ABB RobotStudio station: Solution59_1.rsstn

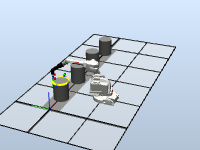
Station Solution59_1 (saved by RobotStudio format 3)
Controller IRB_52_1.20m, task T_ROB1: task frame (RAPID world) sits at (500, 0, 0) mm in the station
Controller IRB_52_1.20m
  mechanical unit CNV1: ?, 1 joints, base frame (0, 0, 0) mm
  mechanical unit ROB_1: IRB52_12_475_1005__01, 6 joints, base frame (500, -1000, 0) mm, rotated rx 0 ry 0 rz 90 deg
Layout (positions relative to the parent item):
  - IRB52_12_475_1005__01 [mechanism, from Robots\IRB52_12_475_1005_G_01.rslib] at (1000, -1000, 0) mm, rotated rx 0 ry 0 rz 90 deg; joint values [0.473, -0.4793, 0.2934, 0.0813, 0.712, -0.0922] (rad or m)
  - Conveyor [conveyor]
    - Part_1 [part]
    - ConveyorObject_31 [conveyorobject] at (3609.02, 0, 0) mm
      - Part_2 [part]
    - ConveyorObject_32 [conveyorobject] at (2609.02, 0, 0) mm
      - Part_2 [part]
    - ConveyorObject_33 [conveyorobject] at (1609.02, 0, 0) mm
      - Part_2 [part]
    - ConveyorObject_34 [conveyorobject] at (609.02, 0, 0) mm
      - Part_2 [part]
  - ROBOBEL926_T_TD_03 [mechanism, from Tools\ROBOBEL926_T_TD_03.rslib] at (734.17, -488.11, 986.41) mm, rotated rx 180 ry 60 rz -59.39 deg
  - Part_2 [part]
Attachment: ROBOBEL926_T_TD_03 is attached to IRB52_12_475_1005__01 / Link6
Conveyor tracking Connection: unit ?, TravelOffset=0.5, QueueTrackDistance=0, StartWindowWidth=1, SyncSeparation=0.1, CountsPerMeter=10000
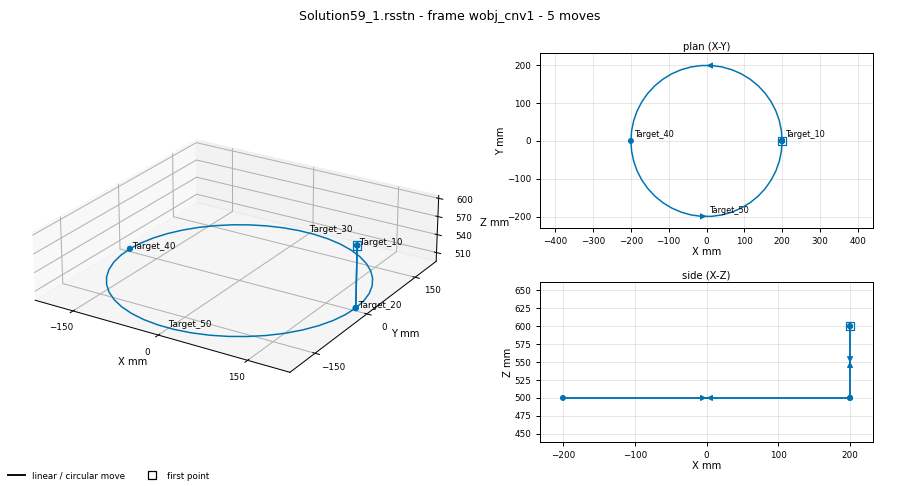
[picture p0: tool path of Solution59_1.rsstn in frame wobj_cnv1, 5 of 7 moves have a stored position in this frame; points joined in program order, loops and branches not executed]
Targets, tools, work objects and paths stored in the station, written as RAPID:
! task T_ROB1
MODULE CalibData
  TASK PERS wobjdata wobj_cnv1:=[FALSE,FALSE,"CNV1",[[0,0,0],[1,0,0,0]],[[0,0,0],[1,0,0,0]]];
  PERS tooldata ROBOBEL926_T_TD_0:=[TRUE,[[117,0,470],[0.866025404,0,0.5,0]],[5.5,[30,0,225],[1,0,0,0],0,0,0]];
  PERS tooldata ROBOBEL926_T_TD_100:=[TRUE,[[204,0,520],[0.866025404,0,0.5,0]],[5.5,[30,0,225],[1,0,0,0],0,0,0]];
  PERS tooldata ROBOBEL926_T_TD_120:=[TRUE,[[220,0,530],[0.866025404,0,0.5,0]],[5.5,[30,0,225],[1,0,0,0],0,0,0]];
  PERS tooldata ROBOBEL926_T_TD_150:=[TRUE,[[247,0,545],[0.866025404,0,0.5,0]],[5.5,[30,0,225],[1,0,0,0],0,0,0]];
  PERS tooldata ROBOBEL926_T_TD_200:=[TRUE,[[290,0,570],[0.866025404,0,0.5,0]],[5.5,[30,0,225],[1,0,0,0],0,0,0]];
  PERS tooldata ROBOBEL926_T_TD_250:=[TRUE,[[333,0,595],[0.866025404,0,0.5,0]],[5.5,[30,0,225],[1,0,0,0],0,0,0]];
  PERS tooldata ROBOBEL926_T_TD_300:=[TRUE,[[377,0,620],[0.866025404,0,0.5,0]],[5.5,[30,0,225],[1,0,0,0],0,0,0]];
ENDMODULE

! task T_ROB1
MODULE Module1
  CONST robtarget Target_10:=[[200,0,600],[0,0.868680579,-0.495372639,0],[-1,0,-1,0],[9E9,9E9,9E9,9E9,9E9,0]];
  CONST robtarget Target_20:=[[200,0,500],[0,0.868680579,-0.495372639,0],[0,0,0,0],[9E9,9E9,9E9,9E9,9E9,0]];
  CONST robtarget Target_30:=[[0,200,500],[0,0.868680579,-0.495372639,0],[0,0,0,0],[9E9,9E9,9E9,9E9,9E9,0]];
  CONST robtarget Target_40:=[[-200,0,500],[0,0.868680579,-0.495372639,0],[0,0,0,0],[9E9,9E9,9E9,9E9,9E9,0]];
  CONST robtarget Target_50:=[[0,-200,500],[0,0.868680579,-0.495372639,0],[0,0,0,0],[9E9,9E9,9E9,9E9,9E9,0]];
  CONST robtarget Target_60:=[[200,0,500],[0,0.868680579,-0.495372639,0],[0,0,0,0],[9E9,9E9,9E9,9E9,9E9,0]];
  CONST robtarget Target_70:=[[200,0,600],[0,0.868680579,-0.495372639,0],[0,0,0,0],[9E9,9E9,9E9,9E9,9E9,0]];
  CONST jointtarget pAbsHome:=[[0,0,0,0,30.000014495,0],[9E9,9E9,9E9,9E9,9E9,0]];
  CONST jointtarget pAbsHome_2:=[[0,0,0,0,30.000014495,0],[9E9,9E9,9E9,9E9,9E9,0]];
  PROC Path_10()
    MoveL Target_10,v1000,z100,ROBOBEL926_T_TD_150\WObj:=wobj_cnv1;
    MoveL Target_20,v1000,z100,ROBOBEL926_T_TD_150\WObj:=wobj_cnv1;
    MoveC Target_30,Target_40,v1000,z100,ROBOBEL926_T_TD_150\WObj:=wobj_cnv1;
    MoveC Target_50,Target_60,v1000,z100,ROBOBEL926_T_TD_150\WObj:=wobj_cnv1;
    MoveL Target_70,v1000,z100,ROBOBEL926_T_TD_150\WObj:=wobj_cnv1;
  ENDPROC
  PROC main2()
    MoveAbsJ pAbsHome,v1000,fine,ROBOBEL926_T_TD_150\WObj:=wobj0;
    ActUnit CNV1;
    WaitWObj wobj_cnv1;
    Path_10;
    MoveAbsJ pAbsHome,v1000,fine,ROBOBEL926_T_TD_150\WObj:=wobj0;
    DropWObj wobj_cnv1;
  ENDPROC
ENDMODULE

